// SIMATIC S7-200 project (STEP 7-Micro/WIN), CPU 224 CN REL 02.01

SYMBOL_TABLE USER1
gio_on_he_thong  VB144    // gio mo he thong
phut_on_he_thong VB145    // phut mo he thong
gio_off_he_thong VB146    // gio tat he thong
phut_off_he_thong VB147    // phut tat he thong
giodautd1        VW666
phutdautd1       VW668
giocuoitd1       VW670
phutcuoitd1      VW672
giodautd2        VW674
phutdautd2       VW676
giocuoitd2       VW678
phutcuoitd2      VW680
giodautd3        VW682
phutdautd3       VW684
giocuoitd3       VW686
phutcuoitd3      VW688
giodautd4        VW690
phutdautd4       VW692
giocuoitd4       VW694
phutcuoitd4      VW696
giodautd5        VW698
phutdautd5       VW700
giocuoitd5       VW702
phutcuoitd5      VW704
giodautd6        VW706
phutdautd6       VW708
giocuoitd6       VW710
phutcuoitd6      VW712
giodautd7        VW714
phutdautd7       VW716
giocuoitd7       VW718
phutcuoitd7      VW720
giodautd8        VW722
phutdautd8       VW724
giocuoitd8       VW726
phutcuoitd8      VW728
t_setup_to_start VW332    // Delay to start
t_xanhtuyen_1    VW200    // thoi gian xanh tuyen 1
t_delayxanhtuyen_1 VW384    // thoi gian delay xanh tuyen 1
t_xanhtuyen_2    VW202    // thoi gian xanh tuyen 2
t_xanhtuyen_3    VW240    // thoi gian xanh tuyen 3
t_vang           VW204    // gia tri thoi gian vang
t_giaitoa        VW206    // thoi gian giai toa xe
t_delay          VW210
t_diboxanhtuyen_3 VW242    // thoi gian di bo xanh tuyen 3
t_tongvangxanht_1 VW320    // thoi gian xanh va vang tuyen 1
t_tongvangxanht_2 VW322    // thoi gian xanh va vang tuyen 2
t_tongvangxanht_3 VW324    // thoi gian xanh va vang tuyen 3
t_tongvangxanht_23 VW326    // thoi gian xanh va vang tuyen 23
t_tongvangxanht_13 VW328    // thoi gian xanh va vang tuyen 13
t_tongvangxanht_12 VW330    // thoi gian xanh va vang tuyen 12
t_gt_xt1         VW212    // t_gt_xt1=thoi gian gt + thoi gian xanh tuyen 1
t_dibodotuyen_1  VW214    // thoi gian di bo do tuyen 1
t_gt_xt2         VW216    // t_gt_xt2=thoi gian gt + thoi gian xanh tuyen 2
t_dibodotuyen_2  VW218    // thoi gian di bo do tuyen 2
t_gt_xt3         VW244    // t_gt_xt3=thoi gian gt + thoi gian xanh tuyen 3
t_dibodotuyen_3  VW246    // thoi gian di bo do tuyen 3
tonggiaitoa1     VW220    // tonggiaitoa1=giaitoa + giaitoa
tonggt1_xt2      VW222    // tonggt1_xt2=tonggiaitoa1+t_xanhtuyen_2
t_dotuyen_1      VW224    // t_dotuyen_1=tonggt_xt2+t_vang
tonggiaitoa2     VW226    // tonggiaitoa2=giaitoa + giaitoa
tonggt1_xt1      VW228    // tonggt1_xt1=tonggiaitoa2+t_xanhtuyen_1
t_dotuyen_2      VW230    // t_dotuyen_2=tonggt_xt1+t_vang
t_dotuyen_3      VW334    // t_dotuyen_2=tonggt_xt1+t_vang
chienluoc_A      M0.0     // bien chien luoc A
chienluoc_B      M0.1     // bien chien luoc B
chienluoc_C      M0.2     // bien chien luoc C
Fmanual          M0.3     // Fmanual
xanhtuyen_1      Q0.0     // ngo ra den xanh tuyen 1
vangtuyen_1      Q0.1     // ngo ra den vang tuyen 1
dotuyen_1        Q0.2     // ngo ra den do tuyen 1
diboxanhtuyen_1  Q0.3     // den xanh nguoi di bo 1
dibodotuyen_1    Q0.4     // den do nguoi di bo tuyen 1
xanhtuyen_2      Q0.5     // ngo ra den xanh tuyen 2
vangtuyen_2      Q0.6     // ngo ra den vang tuyen 2
dotuyen_2        Q0.7     // ngo ra den do tuyen 2
diboxanhtuyen_2  Q1.0     // den di bo xanh tuyen 2
dibodotuyen_2    Q1.1     // den di bo do tuyen 2
dibodotuyen_3    Q2.4     // den do nguoi di bo tuyen 3
diboxanhtuyen_3  Q2.3     // den xanh di bo tuyen 3
dotuyen_3        Q2.2     // ngo ra do tuyen 3
den_db_dem_nguoc Q2.0     // ngo ra den xanh tuyen 3
mui_ten_re       Q2.1     // ngo ra den vang 3
off              I0.0     // kich chop vang
kichtuyen_1      I0.1     // dieu khien tay tuyen 1
kichtuyen_2      I0.2     // dieu khien tay tuyen 2
kichtuyen_3      I0.3     // dieu khien tay tuyen 3
dieu_khien_tay   I0.4     // kich dieu khien tay
nut_bam_di_bo    I0.5     // nut bam di bo
                 ?0_40_0  // vung o nho tam thoi o thoi diem thu 1
t_xanh_t1_td1A   VW20
t_xanh_t2_td1A   VW22
t_xanh_t3_td1A   VW336
t_vang_td1A      VW24
t_giaitoa_t1_td1A VW26
                 ?0_40_0  // vung o nho tam thoi o thoi diem thu 2
t_xanh_t1_td2A   VW30
t_xanh_t2_td2A   VW32
t_xanh_t3_td2A   VW338
t_vang_td2A      VW34
t_giaitoa_t1_td2A VW36
                          // vung o nho tam thoi o thoi diem thu 3
t_xanh_t1_td3A   VW40
t_xanh_t2_td3A   VW42
t_xanh_t3_td3A   VW340
t_vang_td3A      VW44
t_giaitoa_t1_td3A VW46
                          // vung o nho tam thoi o thoi diem thu 4
t_xanh_t1_td4A   VW50
t_xanh_t2_td4A   VW52
t_xanh_t3_td4A   VW342
t_vang_td4A      VW54
t_giaitoa_t1_td4A VW56
                          // vung o nho tam thoi o thoi diem thu 5
t_xanh_t1_td5A   VW60
t_xanh_t2_td5A   VW62
t_xanh_t3_td5A   VW344
t_vang_td5A      VW64
t_giaitoa_t1_td5A VW66
                          // vung o nho tam thoi o thoi diem thu 6
t_xanh_t1_td6A   VW70
t_xanh_t2_td6A   VW72
t_xanh_t3_td6A   VW346
t_vang_td6A      VW74
t_giaitoa_t1_td6A VW76
                          // vung o nho tam thoi o thoi diem thu 7
t_xanh_t1_td7A   VW80
t_xanh_t2_td7A   VW82
t_xanh_t3_td7A   VW348
t_vang_td7A      VW84
t_giaitoa_t1_td7A VW86
                          // vung o nho tam thoi o thoi diem thu 8
t_xanh_t1_td8A   VW312
t_xanh_t2_td8A   VW314
t_xanh_t3_td8A   VW350
t_vang_td8A      VW316
t_giaitoa_t1_td8A VW318
                          // CHIEN LUOC B
                          // vung o nho tam thoi o thoi diem thu 1
t_xanh_t1_td1B   VW88
t_xanh_t2_td1B   VW90
t_xanh_t3_td1B   VW352
t_vang_td1B      VW92
t_giaitoa_t1_td1B VW94
                 ?0_40_0  // vung o nho tam thoi o thoi diem thu 2
t_xanh_t1_td2B   VW96
t_xanh_t2_td2B   VW98
t_xanh_t3_td2B   VW354
t_vang_td2B      VW100
t_giaitoa_t1_td2B VW102
                          // vung o nho tam thoi o thoi diem thu 3
t_xanh_t1_td3B   VW104
t_xanh_t2_td3B   VW106
t_xanh_t3_td3B   VW356
t_vang_td3B      VW108
t_giaitoa_t1_td3B VW110
                          // vung o nho tam thoi o thoi diem thu 4
t_xanh_t1_td4B   VW112
t_xanh_t2_td4B   VW114
t_xanh_t3_td4B   VW358
t_vang_td4B      VW116
t_giaitoa_t1_td4B VW118
                          // vung o nho tam thoi o thoi diem thu 5
t_xanh_t1_td5B   VW120
t_xanh_t2_td5B   VW122
t_xanh_t3_td5B   VW360
t_vang_td5B      VW124
t_giaitoa_t1_td5B VW126
                          // vung o nho tam thoi o thoi diem thu 6
t_xanh_t1_td6B   VW128
t_xanh_t2_td6B   VW130
t_xanh_t3_td6B   VW362
t_vang_td6B      VW132
t_giaitoa_t1_td6B VW134
                          // vung o nho tam thoi o thoi diem thu 7
t_xanh_t1_td7B   VW136
t_xanh_t2_td7B   VW138
t_xanh_t3_td7B   VW364
t_vang_td7B      VW140
t_giaitoa_t1_td7B VW142
                          // vung o nho tam thoi o thoi diem thu 8
t_xanh_t1_td8B   VW232
t_xanh_t2_td8B   VW234
t_xanh_t3_td8B   VW366
t_vang_td8B      VW236
t_giaitoa_t1_td8B VW238
                          // CHIEN LUOC C
                          // vung o nho tam thoi o thoi diem thu 1
t_xanh_t1_td1C   VW248
t_xanh_t2_td1C   VW250
t_xanh_t3_td1C   VW368
t_vang_td1C      VW252
t_giaitoa_t1_td1C VW254
                 ?0_40_0  // vung o nho tam thoi o thoi diem thu 2
t_xanh_t1_td2C   VW256
t_xanh_t2_td2C   VW258
t_xanh_t3_td2C   VW370
t_vang_td2C      VW260
t_giaitoa_t1_td2C VW262
                          // vung o nho tam thoi o thoi diem thu 3
t_xanh_t1_td3C   VW264
t_xanh_t2_td3C   VW266
t_xanh_t3_td3C   VW372
t_vang_td3C      VW268
t_giaitoa_t1_td3C VW270
                          // vung o nho tam thoi o thoi diem thu 4
t_xanh_t1_td4C   VW272
t_xanh_t2_td4C   VW274
t_xanh_t3_td4C   VW374
t_vang_td4C      VW276
t_giaitoa_t1_td4C VW278
                          // vung o nho tam thoi o thoi diem thu 5
t_xanh_t1_td5C   VW280
t_xanh_t2_td5C   VW282
t_xanh_t3_td5C   VW376
t_vang_td5C      VW284
t_giaitoa_t1_td5C VW286
                          // vung o nho tam thoi o thoi diem thu 6
t_xanh_t1_td6C   VW288
t_xanh_t2_td6C   VW290
t_xanh_t3_td6C   VW378
t_vang_td6C      VW292
t_giaitoa_t1_td6C VW294
                          // vung o nho tam thoi o thoi diem thu 7
t_xanh_t1_td7C   VW296
t_xanh_t2_td7C   VW298
t_xanh_t3_td7C   VW380
t_vang_td7C      VW300
t_giaitoa_t1_td7C VW302
                          // vung o nho tam thoi o thoi diem thu 8
t_xanh_t1_td8C   VW304
t_xanh_t2_td8C   VW306
t_xanh_t3_td8C   VW382
t_vang_td8C      VW308
t_giaitoa_t1_td8C VW310
set_time         VB409
set_time_2       VB410
t_phase          VB411
t_dependent      VB412
END_SYMBOL_TABLE

ORGANIZATION_BLOCK MAIN:OB1
TITLE=PROGRAM COMMENTS
BEGIN
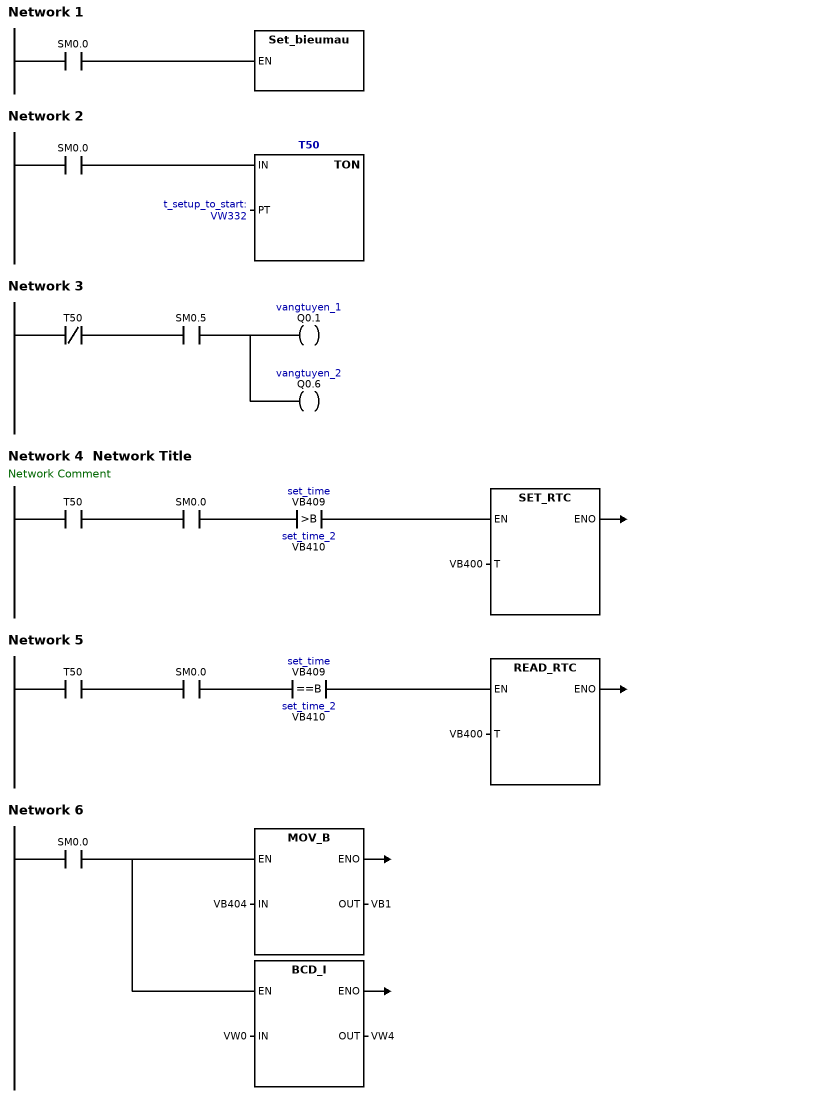
Network 1
LD     SM0.0
CALL   Set_bieumau:SBR18
Network 2
LD     SM0.0
TON    T50, t_setup_to_start:VW332
Network 3
LDN    T50
A      SM0.5
=      vangtuyen_1:Q0.1
=      vangtuyen_2:Q0.6
Network 4 // Network Title
// Network Comment
LD     T50
A      SM0.0
AB>    set_time:VB409, set_time_2:VB410
TODW   VB400
Network 5
LD     T50
A      SM0.0
AB=    set_time:VB409, set_time_2:VB410
TODR   VB400
Network 6
LD     SM0.0
MOVB   VB404, VB1
MOVW   VW0, VW4
BCDI   VW4
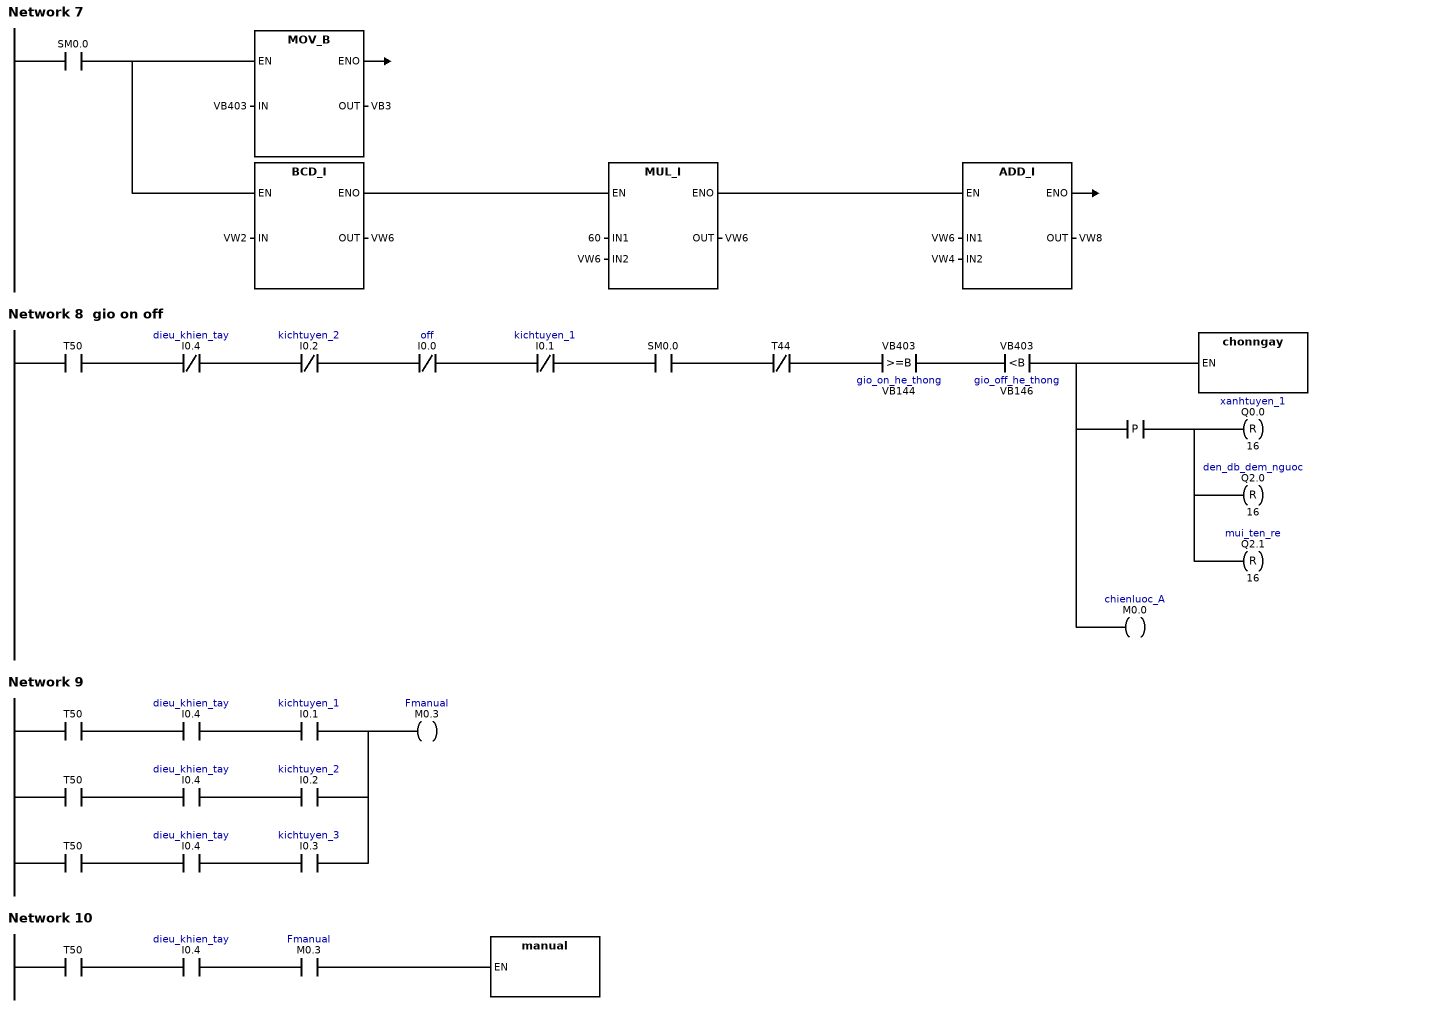
Network 7
LD     SM0.0
MOVB   VB403, VB3
MOVW   VW2, VW6
AENO
BCDI   VW6
AENO
*I     60, VW6
AENO
MOVW   VW6, VW8
+I     VW4, VW8
Network 8 // gio on off
LD     T50
AN     dieu_khien_tay:I0.4
AN     kichtuyen_2:I0.2
AN     off:I0.0
AN     kichtuyen_1:I0.1
A      SM0.0
AN     T44
AB>=   VB403, gio_on_he_thong:VB144
AB<    VB403, gio_off_he_thong:VB146
LPS
CALL   chonngay:SBR11
EU
R      xanhtuyen_1:Q0.0, 16
R      den_db_dem_nguoc:Q2.0, 16
R      mui_ten_re:Q2.1, 16
LPP
=      chienluoc_A:M0.0
Network 9
LD     T50
A      dieu_khien_tay:I0.4
A      kichtuyen_1:I0.1
LD     T50
A      dieu_khien_tay:I0.4
A      kichtuyen_2:I0.2
OLD
LD     T50
A      dieu_khien_tay:I0.4
A      kichtuyen_3:I0.3
OLD
=      Fmanual:M0.3
Network 10
LD     T50
A      dieu_khien_tay:I0.4
A      Fmanual:M0.3
CALL   manual:SBR2
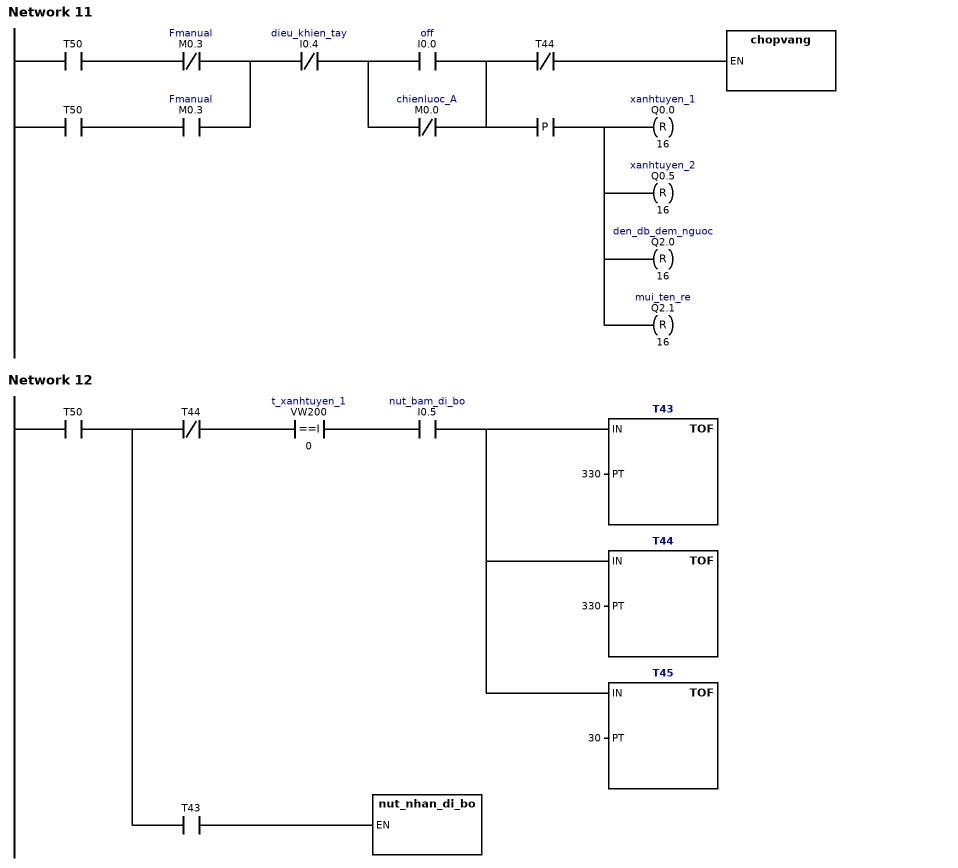
Network 11
LD     T50
AN     Fmanual:M0.3
LD     T50
A      Fmanual:M0.3
OLD
AN     dieu_khien_tay:I0.4
LD     off:I0.0
ON     chienluoc_A:M0.0
ALD
LPS
AN     T44
CALL   chopvang:SBR1
LPP
EU
R      xanhtuyen_1:Q0.0, 16
R      xanhtuyen_2:Q0.5, 16
R      den_db_dem_nguoc:Q2.0, 16
R      mui_ten_re:Q2.1, 16
Network 12
LD     T50
LPS
AN     T44
AW=    t_xanhtuyen_1:VW200, 0
A      nut_bam_di_bo:I0.5
TOF    T43, 330
TOF    T44, 330
TOF    T45, 30
LPP
A      T43
CALL   nut_nhan_di_bo:SBR17
Network 13
// thoi gian giai toa va kich tuyen 2
END_ORGANIZATION_BLOCK

SUBROUTINE_BLOCK tudong2phase:SBR0
TITLE=SUBROUTINE COMMENTS
BEGIN
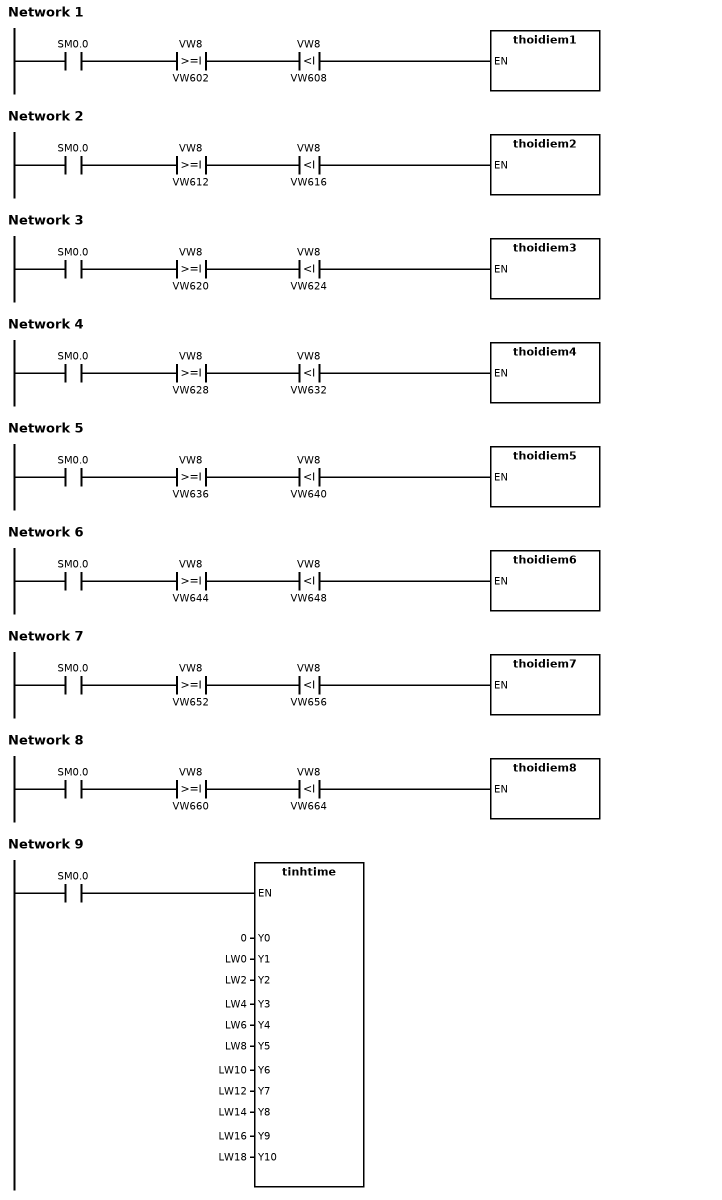
Network 1
LD     SM0.0
AW>=   VW8, VW602
AW<    VW8, VW608
CALL   thoidiem1:SBR3
Network 2
LD     SM0.0
AW>=   VW8, VW612
AW<    VW8, VW616
CALL   thoidiem2:SBR4
Network 3
LD     SM0.0
AW>=   VW8, VW620
AW<    VW8, VW624
CALL   thoidiem3:SBR5
Network 4
LD     SM0.0
AW>=   VW8, VW628
AW<    VW8, VW632
CALL   thoidiem4:SBR6
Network 5
LD     SM0.0
AW>=   VW8, VW636
AW<    VW8, VW640
CALL   thoidiem5:SBR7
Network 6
LD     SM0.0
AW>=   VW8, VW644
AW<    VW8, VW648
CALL   thoidiem6:SBR8
Network 7
LD     SM0.0
AW>=   VW8, VW652
AW<    VW8, VW656
CALL   thoidiem7:SBR9
Network 8
LD     SM0.0
AW>=   VW8, VW660
AW<    VW8, VW664
CALL   thoidiem8:SBR14
Network 9
LD     SM0.0
CALL   tinhtime:SBR16, 0, LW0, LW2, LW4, LW6, LW8, LW10, LW12, LW14, LW16, LW18
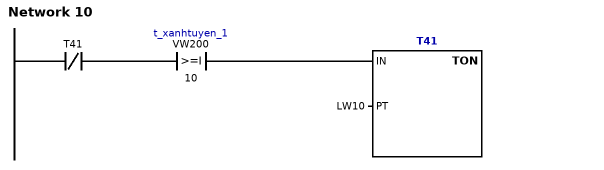
Network 10
LDN    T41
AW>=   t_xanhtuyen_1:VW200, 10
TON    T41, LW10
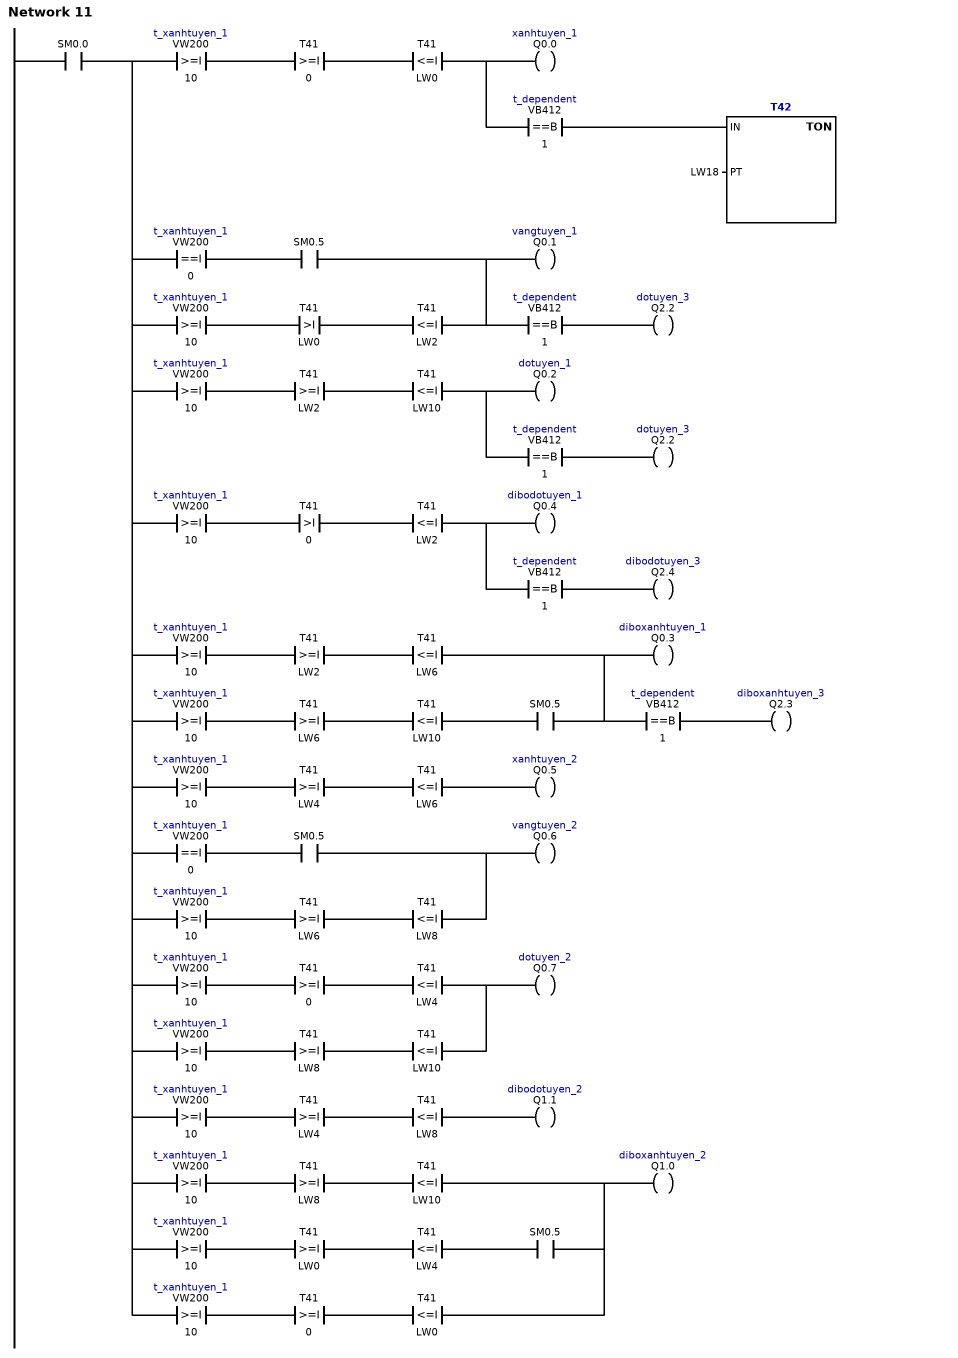
Network 11
LD     SM0.0
LPS
AW>=   t_xanhtuyen_1:VW200, 10
AW>=   T41, 0
AW<=   T41, LW0
=      xanhtuyen_1:Q0.0
AB=    t_dependent:VB412, 1
TON    T42, LW18
LRD
LDW=   t_xanhtuyen_1:VW200, 0
A      SM0.5
LDW>=  t_xanhtuyen_1:VW200, 10
AW>    T41, LW0
AW<=   T41, LW2
OLD
ALD
=      vangtuyen_1:Q0.1
AB=    t_dependent:VB412, 1
=      dotuyen_3:Q2.2
LRD
AW>=   t_xanhtuyen_1:VW200, 10
AW>=   T41, LW2
AW<=   T41, LW10
=      dotuyen_1:Q0.2
AB=    t_dependent:VB412, 1
=      dotuyen_3:Q2.2
LRD
AW>=   t_xanhtuyen_1:VW200, 10
AW>    T41, 0
AW<=   T41, LW2
=      dibodotuyen_1:Q0.4
AB=    t_dependent:VB412, 1
=      dibodotuyen_3:Q2.4
LRD
LDW>=  t_xanhtuyen_1:VW200, 10
AW>=   T41, LW2
AW<=   T41, LW6
LDW>=  t_xanhtuyen_1:VW200, 10
AW>=   T41, LW6
AW<=   T41, LW10
A      SM0.5
OLD
ALD
=      diboxanhtuyen_1:Q0.3
AB=    t_dependent:VB412, 1
=      diboxanhtuyen_3:Q2.3
LRD
AW>=   t_xanhtuyen_1:VW200, 10
AW>=   T41, LW4
AW<=   T41, LW6
=      xanhtuyen_2:Q0.5
LRD
LDW=   t_xanhtuyen_1:VW200, 0
A      SM0.5
LDW>=  t_xanhtuyen_1:VW200, 10
AW>=   T41, LW6
AW<=   T41, LW8
OLD
ALD
=      vangtuyen_2:Q0.6
LRD
LDW>=  t_xanhtuyen_1:VW200, 10
AW>=   T41, 0
AW<=   T41, LW4
LDW>=  t_xanhtuyen_1:VW200, 10
AW>=   T41, LW8
AW<=   T41, LW10
OLD
ALD
=      dotuyen_2:Q0.7
LRD
AW>=   t_xanhtuyen_1:VW200, 10
AW>=   T41, LW4
AW<=   T41, LW8
=      dibodotuyen_2:Q1.1
LPP
LDW>=  t_xanhtuyen_1:VW200, 10
AW>=   T41, LW8
AW<=   T41, LW10
LDW>=  t_xanhtuyen_1:VW200, 10
AW>=   T41, LW0
AW<=   T41, LW4
A      SM0.5
OLD
LDW>=  t_xanhtuyen_1:VW200, 10
AW>=   T41, 0
AW<=   T41, LW0
OLD
ALD
=      diboxanhtuyen_2:Q1.0
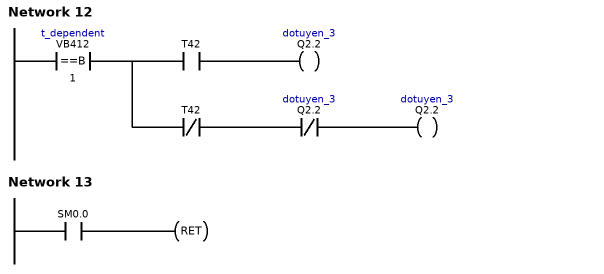
Network 12
LDB=   t_dependent:VB412, 1
LPS
A      T42
=      dotuyen_3:Q2.2
LPP
AN     T42
AN     dotuyen_3:Q2.2
=      dotuyen_3:Q2.2
Network 13
LD     SM0.0
CRET
END_SUBROUTINE_BLOCK

SUBROUTINE_BLOCK chopvang:SBR1
TITLE=SUBROUTINE COMMENTS
BEGIN
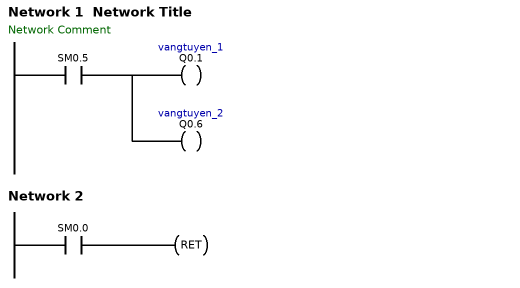
Network 1 // Network Title
// Network Comment
LD     SM0.5
=      vangtuyen_1:Q0.1
=      vangtuyen_2:Q0.6
Network 2
LD     SM0.0
CRET
END_SUBROUTINE_BLOCK

SUBROUTINE_BLOCK manual:SBR2
TITLE=SUBROUTINE COMMENTS
BEGIN
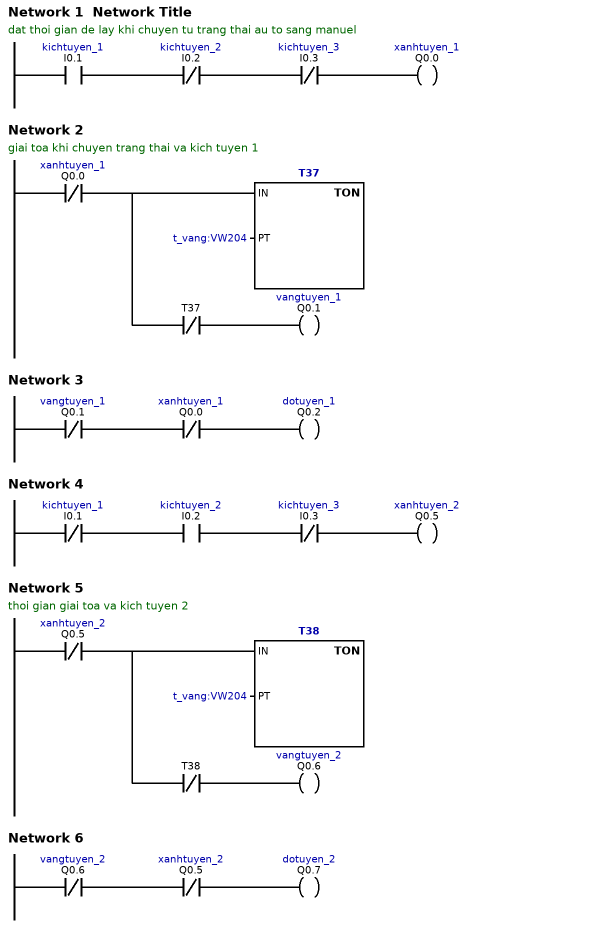
Network 1 // Network Title
// dat thoi gian de lay khi chuyen tu trang thai au to sang manuel
LD     kichtuyen_1:I0.1
AN     kichtuyen_2:I0.2
AN     kichtuyen_3:I0.3
=      xanhtuyen_1:Q0.0
Network 2
// giai toa khi chuyen trang thai va kich tuyen 1
LDN    xanhtuyen_1:Q0.0
TON    T37, t_vang:VW204
AN     T37
=      vangtuyen_1:Q0.1
Network 3
LDN    vangtuyen_1:Q0.1
AN     xanhtuyen_1:Q0.0
=      dotuyen_1:Q0.2
Network 4
LDN    kichtuyen_1:I0.1
A      kichtuyen_2:I0.2
AN     kichtuyen_3:I0.3
=      xanhtuyen_2:Q0.5
Network 5
// thoi gian giai toa va kich tuyen 2
LDN    xanhtuyen_2:Q0.5
TON    T38, t_vang:VW204
AN     T38
=      vangtuyen_2:Q0.6
Network 6
LDN    vangtuyen_2:Q0.6
AN     xanhtuyen_2:Q0.5
=      dotuyen_2:Q0.7
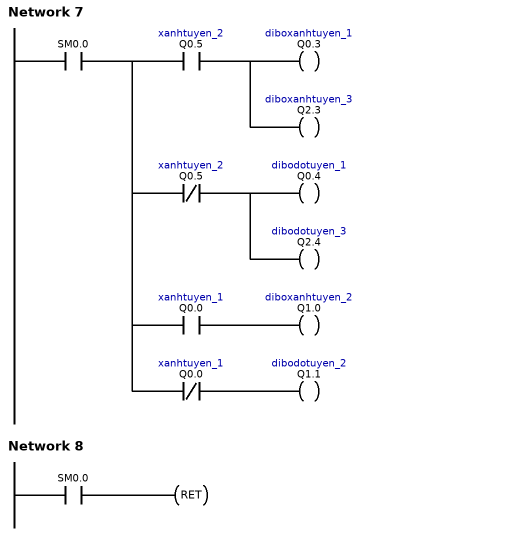
Network 7
LD     SM0.0
LPS
A      xanhtuyen_2:Q0.5
=      diboxanhtuyen_1:Q0.3
=      diboxanhtuyen_3:Q2.3
LRD
AN     xanhtuyen_2:Q0.5
=      dibodotuyen_1:Q0.4
=      dibodotuyen_3:Q2.4
LPP
LPS
A      xanhtuyen_1:Q0.0
=      diboxanhtuyen_2:Q1.0
LPP
AN     xanhtuyen_1:Q0.0
=      dibodotuyen_2:Q1.1
Network 8
LD     SM0.0
CRET
END_SUBROUTINE_BLOCK

SUBROUTINE_BLOCK thoidiem1:SBR3
TITLE=SUBROUTINE COMMENTS
BEGIN
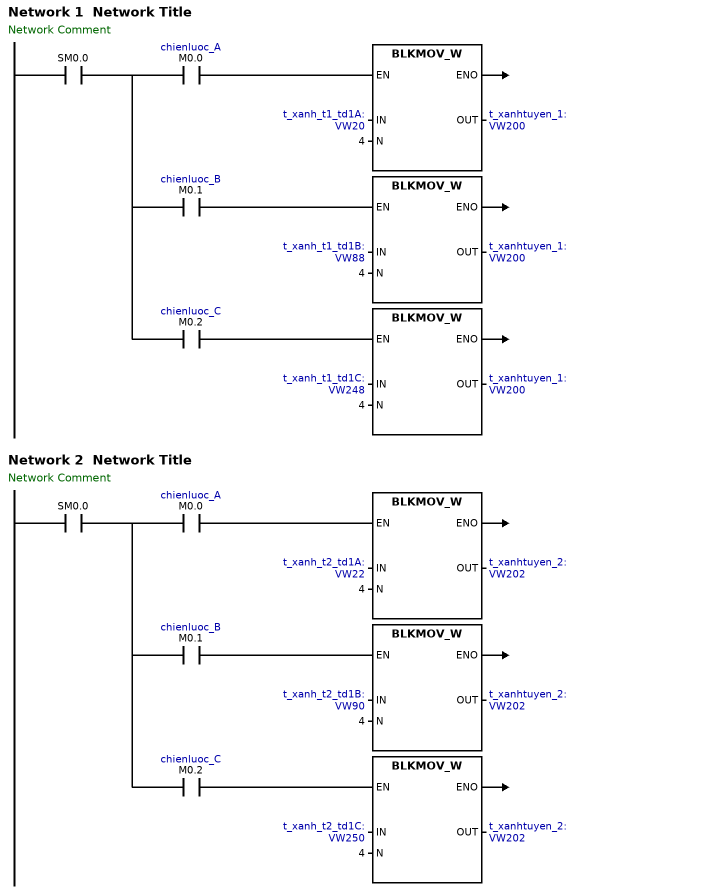
Network 1 // Network Title
// Network Comment
LD     SM0.0
LPS
A      chienluoc_A:M0.0
BMW    t_xanh_t1_td1A:VW20, t_xanhtuyen_1:VW200, 4
LRD
A      chienluoc_B:M0.1
BMW    t_xanh_t1_td1B:VW88, t_xanhtuyen_1:VW200, 4
LPP
A      chienluoc_C:M0.2
BMW    t_xanh_t1_td1C:VW248, t_xanhtuyen_1:VW200, 4
Network 2 // Network Title
// Network Comment
LD     SM0.0
LPS
A      chienluoc_A:M0.0
BMW    t_xanh_t2_td1A:VW22, t_xanhtuyen_2:VW202, 4
LRD
A      chienluoc_B:M0.1
BMW    t_xanh_t2_td1B:VW90, t_xanhtuyen_2:VW202, 4
LPP
A      chienluoc_C:M0.2
BMW    t_xanh_t2_td1C:VW250, t_xanhtuyen_2:VW202, 4
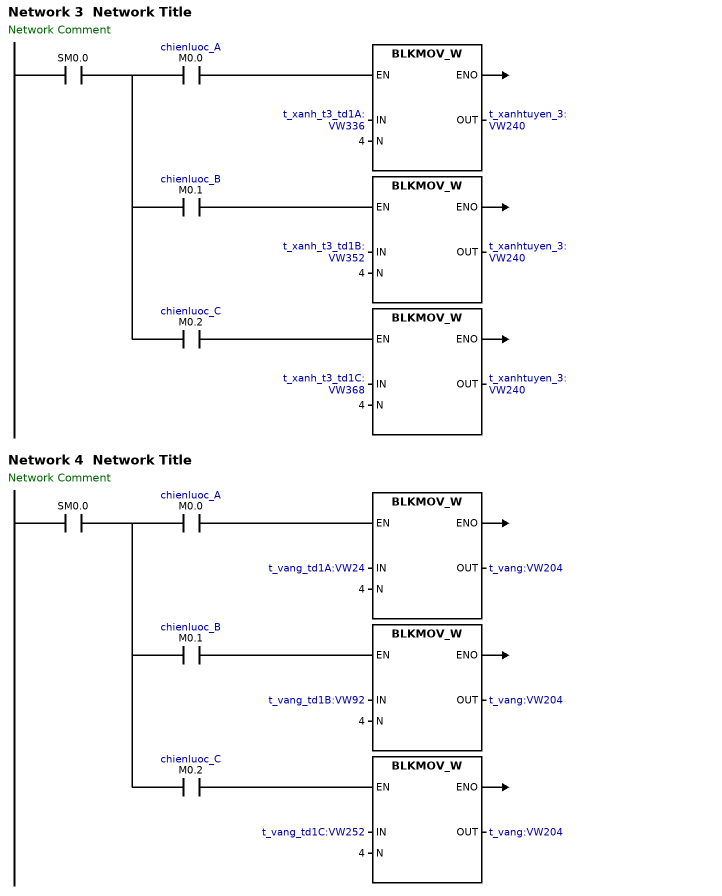
Network 3 // Network Title
// Network Comment
LD     SM0.0
LPS
A      chienluoc_A:M0.0
BMW    t_xanh_t3_td1A:VW336, t_xanhtuyen_3:VW240, 4
LRD
A      chienluoc_B:M0.1
BMW    t_xanh_t3_td1B:VW352, t_xanhtuyen_3:VW240, 4
LPP
A      chienluoc_C:M0.2
BMW    t_xanh_t3_td1C:VW368, t_xanhtuyen_3:VW240, 4
Network 4 // Network Title
// Network Comment
LD     SM0.0
LPS
A      chienluoc_A:M0.0
BMW    t_vang_td1A:VW24, t_vang:VW204, 4
LRD
A      chienluoc_B:M0.1
BMW    t_vang_td1B:VW92, t_vang:VW204, 4
LPP
A      chienluoc_C:M0.2
BMW    t_vang_td1C:VW252, t_vang:VW204, 4
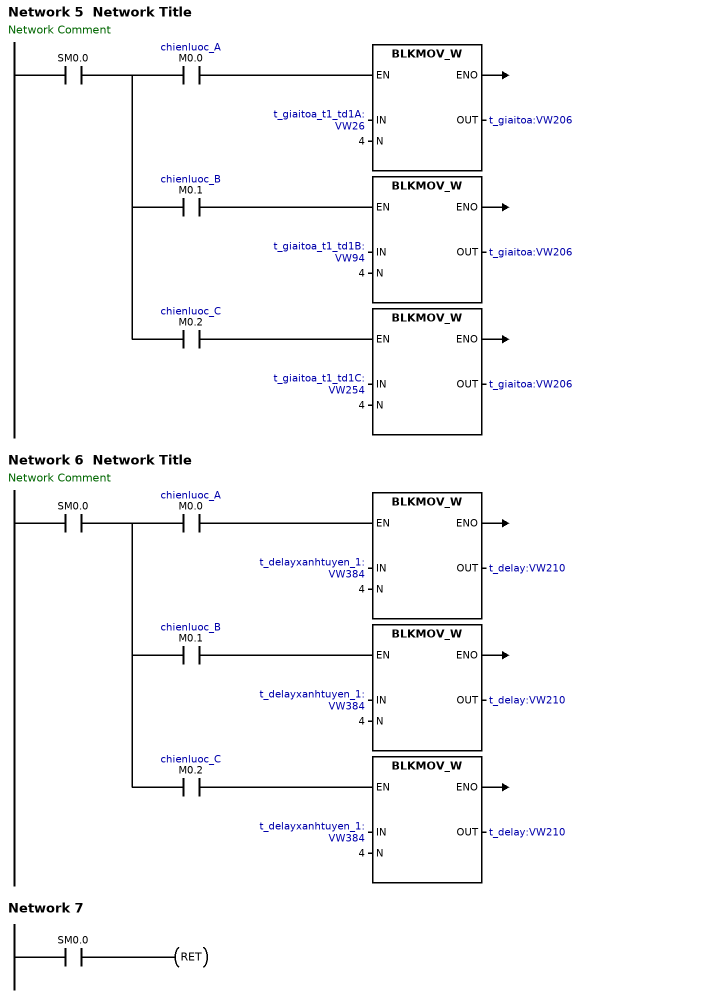
Network 5 // Network Title
// Network Comment
LD     SM0.0
LPS
A      chienluoc_A:M0.0
BMW    t_giaitoa_t1_td1A:VW26, t_giaitoa:VW206, 4
LRD
A      chienluoc_B:M0.1
BMW    t_giaitoa_t1_td1B:VW94, t_giaitoa:VW206, 4
LPP
A      chienluoc_C:M0.2
BMW    t_giaitoa_t1_td1C:VW254, t_giaitoa:VW206, 4
Network 6 // Network Title
// Network Comment
LD     SM0.0
LPS
A      chienluoc_A:M0.0
BMW    t_delayxanhtuyen_1:VW384, t_delay:VW210, 4
LRD
A      chienluoc_B:M0.1
BMW    t_delayxanhtuyen_1:VW384, t_delay:VW210, 4
LPP
A      chienluoc_C:M0.2
BMW    t_delayxanhtuyen_1:VW384, t_delay:VW210, 4
Network 7
LD     SM0.0
CRET
END_SUBROUTINE_BLOCK

SUBROUTINE_BLOCK thoidiem2:SBR4
TITLE=SUBROUTINE COMMENTS
BEGIN
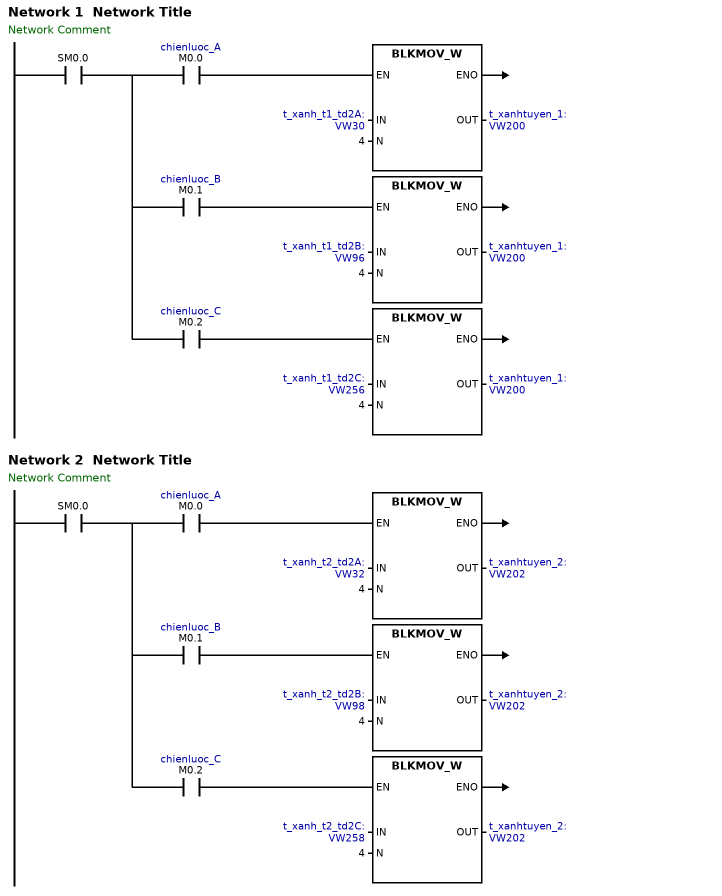
Network 1 // Network Title
// Network Comment
LD     SM0.0
LPS
A      chienluoc_A:M0.0
BMW    t_xanh_t1_td2A:VW30, t_xanhtuyen_1:VW200, 4
LRD
A      chienluoc_B:M0.1
BMW    t_xanh_t1_td2B:VW96, t_xanhtuyen_1:VW200, 4
LPP
A      chienluoc_C:M0.2
BMW    t_xanh_t1_td2C:VW256, t_xanhtuyen_1:VW200, 4
Network 2 // Network Title
// Network Comment
LD     SM0.0
LPS
A      chienluoc_A:M0.0
BMW    t_xanh_t2_td2A:VW32, t_xanhtuyen_2:VW202, 4
LRD
A      chienluoc_B:M0.1
BMW    t_xanh_t2_td2B:VW98, t_xanhtuyen_2:VW202, 4
LPP
A      chienluoc_C:M0.2
BMW    t_xanh_t2_td2C:VW258, t_xanhtuyen_2:VW202, 4
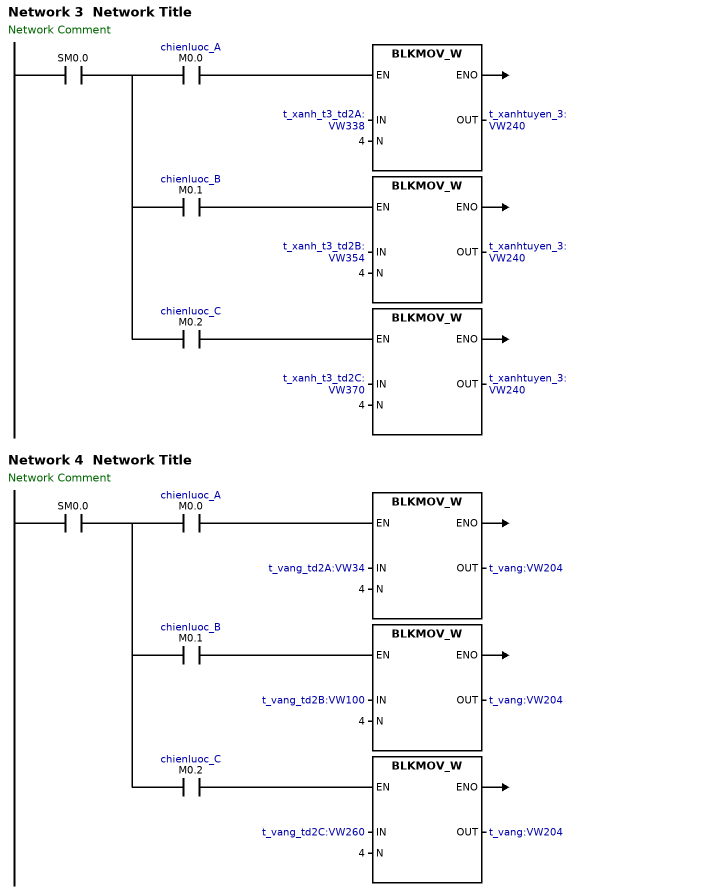
Network 3 // Network Title
// Network Comment
LD     SM0.0
LPS
A      chienluoc_A:M0.0
BMW    t_xanh_t3_td2A:VW338, t_xanhtuyen_3:VW240, 4
LRD
A      chienluoc_B:M0.1
BMW    t_xanh_t3_td2B:VW354, t_xanhtuyen_3:VW240, 4
LPP
A      chienluoc_C:M0.2
BMW    t_xanh_t3_td2C:VW370, t_xanhtuyen_3:VW240, 4
Network 4 // Network Title
// Network Comment
LD     SM0.0
LPS
A      chienluoc_A:M0.0
BMW    t_vang_td2A:VW34, t_vang:VW204, 4
LRD
A      chienluoc_B:M0.1
BMW    t_vang_td2B:VW100, t_vang:VW204, 4
LPP
A      chienluoc_C:M0.2
BMW    t_vang_td2C:VW260, t_vang:VW204, 4
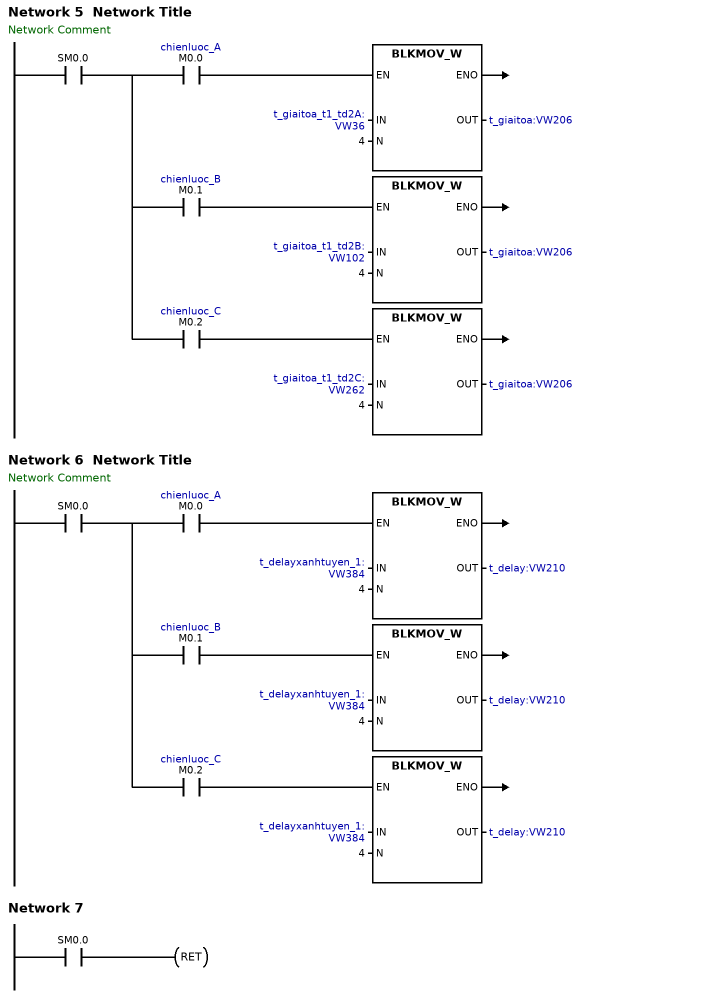
Network 5 // Network Title
// Network Comment
LD     SM0.0
LPS
A      chienluoc_A:M0.0
BMW    t_giaitoa_t1_td2A:VW36, t_giaitoa:VW206, 4
LRD
A      chienluoc_B:M0.1
BMW    t_giaitoa_t1_td2B:VW102, t_giaitoa:VW206, 4
LPP
A      chienluoc_C:M0.2
BMW    t_giaitoa_t1_td2C:VW262, t_giaitoa:VW206, 4
Network 6 // Network Title
// Network Comment
LD     SM0.0
LPS
A      chienluoc_A:M0.0
BMW    t_delayxanhtuyen_1:VW384, t_delay:VW210, 4
LRD
A      chienluoc_B:M0.1
BMW    t_delayxanhtuyen_1:VW384, t_delay:VW210, 4
LPP
A      chienluoc_C:M0.2
BMW    t_delayxanhtuyen_1:VW384, t_delay:VW210, 4
Network 7
LD     SM0.0
CRET
END_SUBROUTINE_BLOCK

SUBROUTINE_BLOCK thoidiem3:SBR5
TITLE=SUBROUTINE COMMENTS
BEGIN
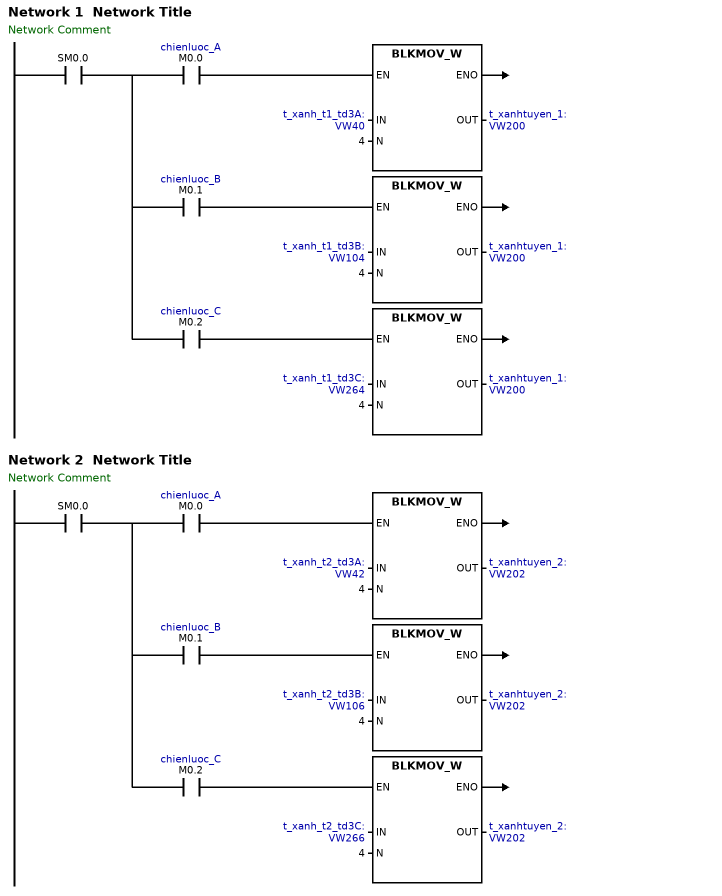
Network 1 // Network Title
// Network Comment
LD     SM0.0
LPS
A      chienluoc_A:M0.0
BMW    t_xanh_t1_td3A:VW40, t_xanhtuyen_1:VW200, 4
LRD
A      chienluoc_B:M0.1
BMW    t_xanh_t1_td3B:VW104, t_xanhtuyen_1:VW200, 4
LPP
A      chienluoc_C:M0.2
BMW    t_xanh_t1_td3C:VW264, t_xanhtuyen_1:VW200, 4
Network 2 // Network Title
// Network Comment
LD     SM0.0
LPS
A      chienluoc_A:M0.0
BMW    t_xanh_t2_td3A:VW42, t_xanhtuyen_2:VW202, 4
LRD
A      chienluoc_B:M0.1
BMW    t_xanh_t2_td3B:VW106, t_xanhtuyen_2:VW202, 4
LPP
A      chienluoc_C:M0.2
BMW    t_xanh_t2_td3C:VW266, t_xanhtuyen_2:VW202, 4
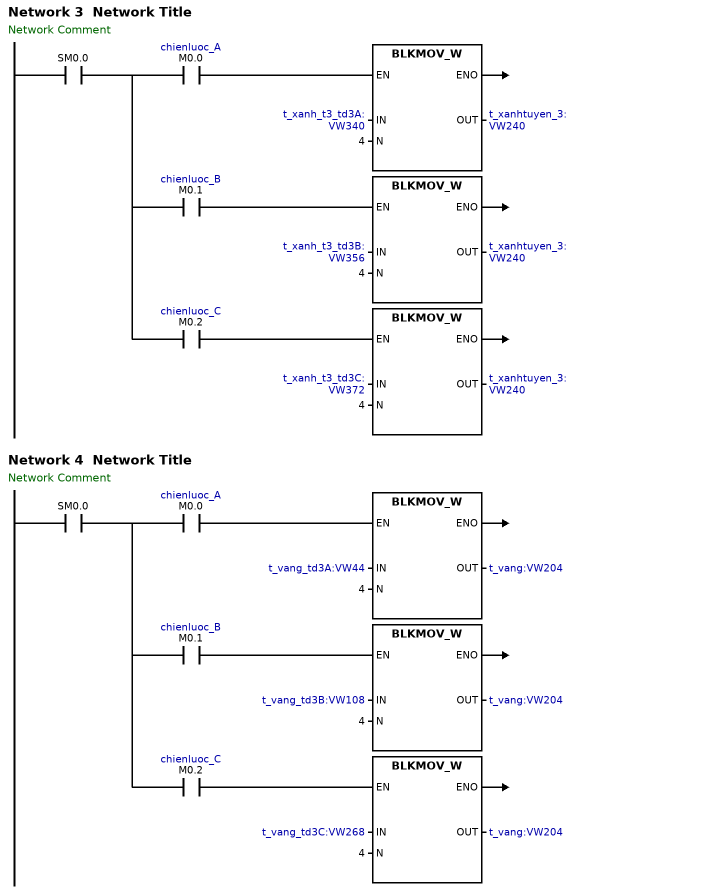
Network 3 // Network Title
// Network Comment
LD     SM0.0
LPS
A      chienluoc_A:M0.0
BMW    t_xanh_t3_td3A:VW340, t_xanhtuyen_3:VW240, 4
LRD
A      chienluoc_B:M0.1
BMW    t_xanh_t3_td3B:VW356, t_xanhtuyen_3:VW240, 4
LPP
A      chienluoc_C:M0.2
BMW    t_xanh_t3_td3C:VW372, t_xanhtuyen_3:VW240, 4
Network 4 // Network Title
// Network Comment
LD     SM0.0
LPS
A      chienluoc_A:M0.0
BMW    t_vang_td3A:VW44, t_vang:VW204, 4
LRD
A      chienluoc_B:M0.1
BMW    t_vang_td3B:VW108, t_vang:VW204, 4
LPP
A      chienluoc_C:M0.2
BMW    t_vang_td3C:VW268, t_vang:VW204, 4
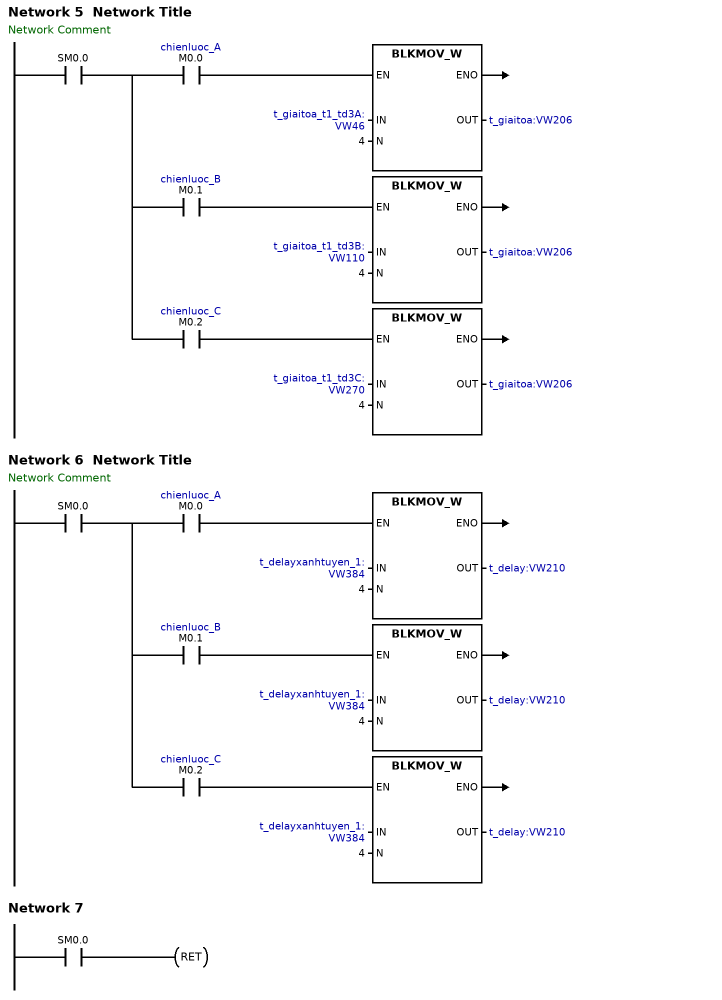
Network 5 // Network Title
// Network Comment
LD     SM0.0
LPS
A      chienluoc_A:M0.0
BMW    t_giaitoa_t1_td3A:VW46, t_giaitoa:VW206, 4
LRD
A      chienluoc_B:M0.1
BMW    t_giaitoa_t1_td3B:VW110, t_giaitoa:VW206, 4
LPP
A      chienluoc_C:M0.2
BMW    t_giaitoa_t1_td3C:VW270, t_giaitoa:VW206, 4
Network 6 // Network Title
// Network Comment
LD     SM0.0
LPS
A      chienluoc_A:M0.0
BMW    t_delayxanhtuyen_1:VW384, t_delay:VW210, 4
LRD
A      chienluoc_B:M0.1
BMW    t_delayxanhtuyen_1:VW384, t_delay:VW210, 4
LPP
A      chienluoc_C:M0.2
BMW    t_delayxanhtuyen_1:VW384, t_delay:VW210, 4
Network 7
LD     SM0.0
CRET
END_SUBROUTINE_BLOCK

SUBROUTINE_BLOCK thoidiem4:SBR6
TITLE=SUBROUTINE COMMENTS
BEGIN
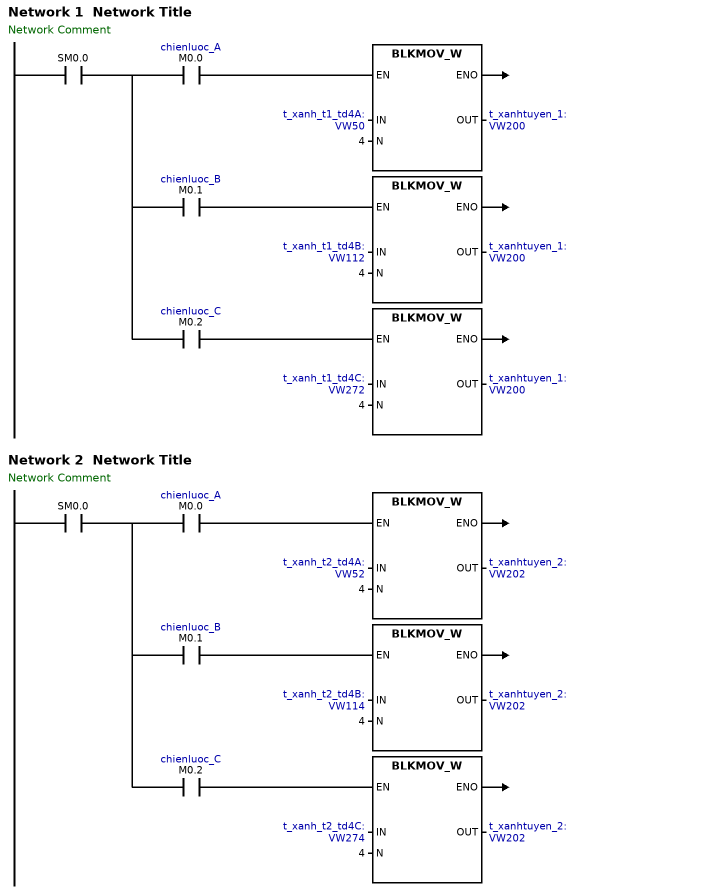
Network 1 // Network Title
// Network Comment
LD     SM0.0
LPS
A      chienluoc_A:M0.0
BMW    t_xanh_t1_td4A:VW50, t_xanhtuyen_1:VW200, 4
LRD
A      chienluoc_B:M0.1
BMW    t_xanh_t1_td4B:VW112, t_xanhtuyen_1:VW200, 4
LPP
A      chienluoc_C:M0.2
BMW    t_xanh_t1_td4C:VW272, t_xanhtuyen_1:VW200, 4
Network 2 // Network Title
// Network Comment
LD     SM0.0
LPS
A      chienluoc_A:M0.0
BMW    t_xanh_t2_td4A:VW52, t_xanhtuyen_2:VW202, 4
LRD
A      chienluoc_B:M0.1
BMW    t_xanh_t2_td4B:VW114, t_xanhtuyen_2:VW202, 4
LPP
A      chienluoc_C:M0.2
BMW    t_xanh_t2_td4C:VW274, t_xanhtuyen_2:VW202, 4
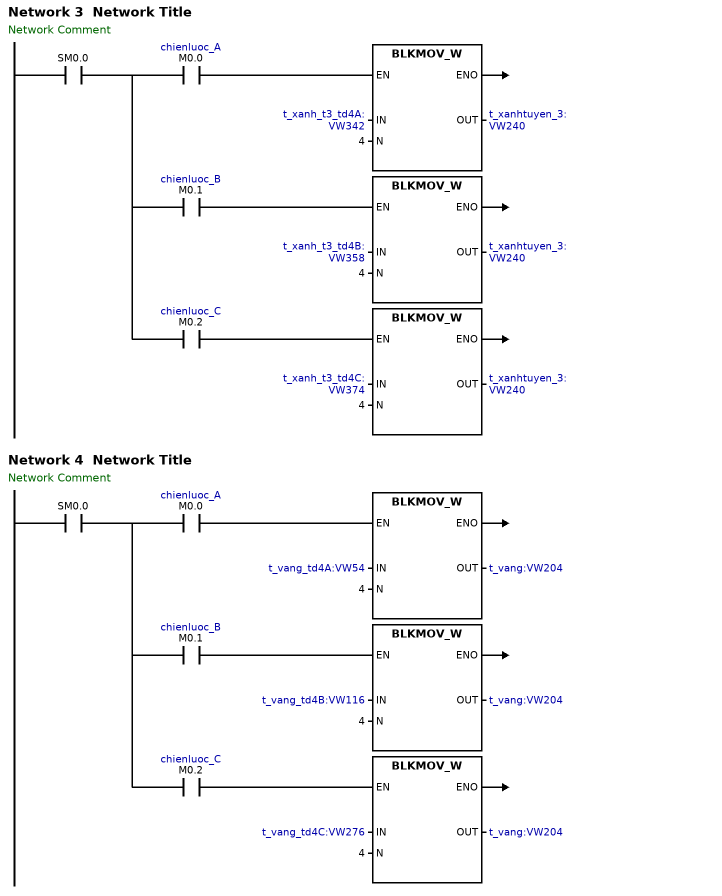
Network 3 // Network Title
// Network Comment
LD     SM0.0
LPS
A      chienluoc_A:M0.0
BMW    t_xanh_t3_td4A:VW342, t_xanhtuyen_3:VW240, 4
LRD
A      chienluoc_B:M0.1
BMW    t_xanh_t3_td4B:VW358, t_xanhtuyen_3:VW240, 4
LPP
A      chienluoc_C:M0.2
BMW    t_xanh_t3_td4C:VW374, t_xanhtuyen_3:VW240, 4
Network 4 // Network Title
// Network Comment
LD     SM0.0
LPS
A      chienluoc_A:M0.0
BMW    t_vang_td4A:VW54, t_vang:VW204, 4
LRD
A      chienluoc_B:M0.1
BMW    t_vang_td4B:VW116, t_vang:VW204, 4
LPP
A      chienluoc_C:M0.2
BMW    t_vang_td4C:VW276, t_vang:VW204, 4
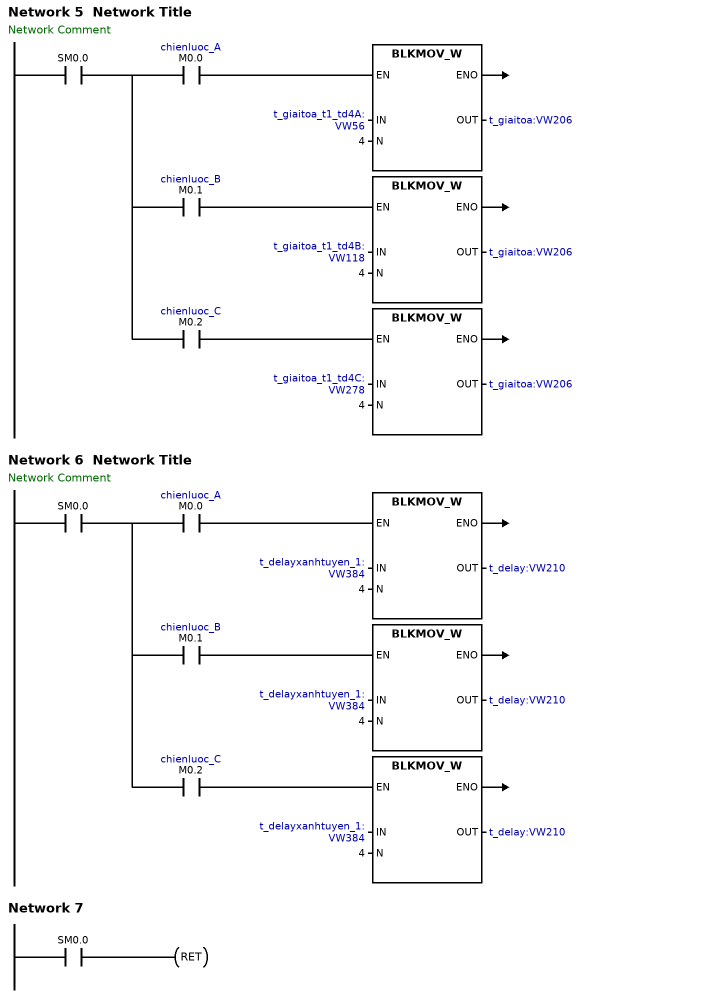
Network 5 // Network Title
// Network Comment
LD     SM0.0
LPS
A      chienluoc_A:M0.0
BMW    t_giaitoa_t1_td4A:VW56, t_giaitoa:VW206, 4
LRD
A      chienluoc_B:M0.1
BMW    t_giaitoa_t1_td4B:VW118, t_giaitoa:VW206, 4
LPP
A      chienluoc_C:M0.2
BMW    t_giaitoa_t1_td4C:VW278, t_giaitoa:VW206, 4
Network 6 // Network Title
// Network Comment
LD     SM0.0
LPS
A      chienluoc_A:M0.0
BMW    t_delayxanhtuyen_1:VW384, t_delay:VW210, 4
LRD
A      chienluoc_B:M0.1
BMW    t_delayxanhtuyen_1:VW384, t_delay:VW210, 4
LPP
A      chienluoc_C:M0.2
BMW    t_delayxanhtuyen_1:VW384, t_delay:VW210, 4
Network 7
LD     SM0.0
CRET
END_SUBROUTINE_BLOCK

SUBROUTINE_BLOCK thoidiem5:SBR7
TITLE=SUBROUTINE COMMENTS
BEGIN
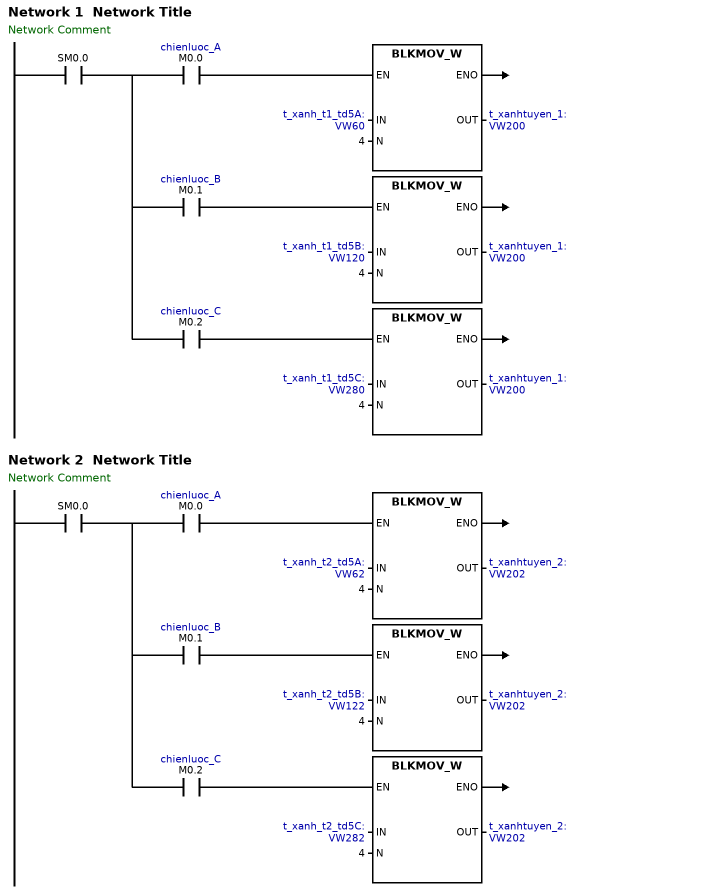
Network 1 // Network Title
// Network Comment
LD     SM0.0
LPS
A      chienluoc_A:M0.0
BMW    t_xanh_t1_td5A:VW60, t_xanhtuyen_1:VW200, 4
LRD
A      chienluoc_B:M0.1
BMW    t_xanh_t1_td5B:VW120, t_xanhtuyen_1:VW200, 4
LPP
A      chienluoc_C:M0.2
BMW    t_xanh_t1_td5C:VW280, t_xanhtuyen_1:VW200, 4
Network 2 // Network Title
// Network Comment
LD     SM0.0
LPS
A      chienluoc_A:M0.0
BMW    t_xanh_t2_td5A:VW62, t_xanhtuyen_2:VW202, 4
LRD
A      chienluoc_B:M0.1
BMW    t_xanh_t2_td5B:VW122, t_xanhtuyen_2:VW202, 4
LPP
A      chienluoc_C:M0.2
BMW    t_xanh_t2_td5C:VW282, t_xanhtuyen_2:VW202, 4
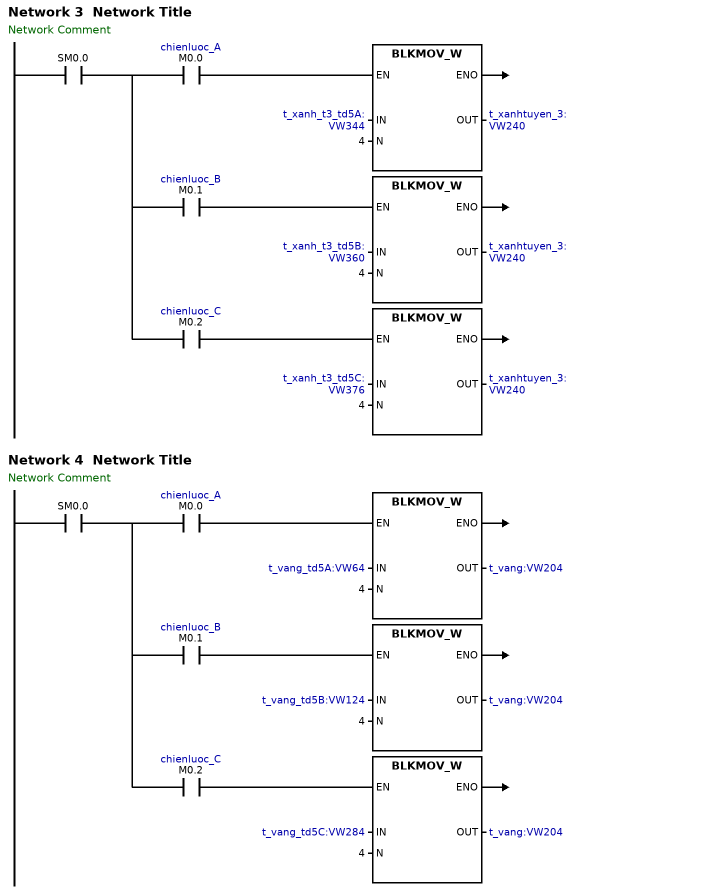
Network 3 // Network Title
// Network Comment
LD     SM0.0
LPS
A      chienluoc_A:M0.0
BMW    t_xanh_t3_td5A:VW344, t_xanhtuyen_3:VW240, 4
LRD
A      chienluoc_B:M0.1
BMW    t_xanh_t3_td5B:VW360, t_xanhtuyen_3:VW240, 4
LPP
A      chienluoc_C:M0.2
BMW    t_xanh_t3_td5C:VW376, t_xanhtuyen_3:VW240, 4
Network 4 // Network Title
// Network Comment
LD     SM0.0
LPS
A      chienluoc_A:M0.0
BMW    t_vang_td5A:VW64, t_vang:VW204, 4
LRD
A      chienluoc_B:M0.1
BMW    t_vang_td5B:VW124, t_vang:VW204, 4
LPP
A      chienluoc_C:M0.2
BMW    t_vang_td5C:VW284, t_vang:VW204, 4
